INTERFACE Istate

METHOD mExecute
VAR_INPUT
END_VAR
END_METHOD

METHOD mHold
VAR_INPUT
END_VAR
END_METHOD

METHOD mStart
VAR_INPUT
END_VAR
END_METHOD

METHOD mStop
VAR_INPUT
END_VAR
END_METHOD

PROPERTY pMessage : String
GET
END_GET
END_PROPERTY

END_INTERFACE

(* stored: Version 1.1.0.1, ProductVersion 3.1.4024.9
   Itf Istate: Id {abd74a6c-8f35-442c-b708-0cd9d237a262}
   Method mExecute: Id {16b552e6-1a3a-498d-934a-985d1bae9d2f}
   Method mHold: Id {b92f87df-f37e-4730-b35d-a3120e980482}
   Method mStart: Id {4cd822d5-9850-4987-90c0-28d3dd087088}
   Method mStop: Id {b1f20e9f-24a3-44e8-a918-984751cd0d27}
   Property pMessage: Id {65b2abd4-9067-42b8-b38b-5c3000e721dc}
   Get Get: Id {e6666da1-b2ef-41c0-b993-79e7fef66188} *)
